Universal Robots PolyScope program: a_full_bow.urp

Program a_full_bow (installation=string_planes directory=/programs createdIn=5.17.3 lastSavedIn=5.17.3 robotSerialNumber=20245501435)
Calibrated DH parameters: a=[0.000154, -0.137004, -0.385524, -0.00002, 0.000092, 0]; d=[0.162441, 211.794786, -230.585024, 18.923638, 0.099786, 0.09951]; alpha=[1.569493, -0.001902, 0.003874, 1.570111, -1.570167, 0]; deltaTheta=[0, -1.242934, 1.056292, 0.186646, 0.000002, 0.000001]
InitVariablesNode
Robot Program (runOnlyOnce=false)
  bow_dir := False
  note_dur := 3
  Timer (action=Start) variable(name=timer_1)
  If bow_dir
    MoveL speed 250 mm/s, acceleration 1200 mm/s^2 (useActiveTCP=true) feature=Base
      Waypoint Waypoint_2: TCP in base x=374.969 y=359.127 z=303.035 mm, rx=1.6275 ry=2.3373 rz=-1.1146 rad; joints [-156.117, -66.368, 101.552, -88.734, -114.429, -168.118] deg; TCP offset x=28.21 y=-96.107 z=-99.69 mm, rx=0 ry=0 rz=0 rad
        Until EXPRESSION (allowActions=false) ExpressionBranch=timer_1≟note_dur
  Else 
    MoveL speed 250 mm/s, acceleration 1200 mm/s^2 (useActiveTCP=true) feature=Base
      Waypoint Waypoint_1: TCP in base x=277.237 y=734.032 z=156.892 mm, rx=1.7389 ry=2.3104 rz=-1.1078 rad; joints [-126.647, -28.123, 54.729, -74.616, -91.964, -141.812] deg; TCP offset x=28.21 y=-96.107 z=-99.69 mm, rx=0 ry=0 rz=0 rad
        Until EXPRESSION (allowActions=false) ExpressionBranch=timer_1≟note_dur
  SuppressedNode
    MoveL speed 250 mm/s, acceleration 1200 mm/s^2 (useActiveTCP=true) feature=Base
      Waypoint Waypoint_1: TCP in base x=277.237 y=734.032 z=156.892 mm, rx=1.7389 ry=2.3104 rz=-1.1078 rad; joints [-126.647, -28.123, 54.729, -74.616, -91.964, -141.812] deg
      Waypoint Waypoint_3: motionParameters(blendRadius=0.05); TCP in base x=335.809 y=527.638 z=230.762 mm, rx=1.7389 ry=2.3104 rz=-1.1078 rad; joints [-141.244, -51.172, 87.867, -86.053, -101.589, -152.842] deg; TCP offset x=28.21 y=-96.107 z=-99.69 mm, rx=0 ry=0 rz=0 rad
      Waypoint Waypoint_2: TCP in base x=393.128 y=325.659 z=303.053 mm, rx=1.7389 ry=2.3104 rz=-1.1078 rad; joints [-160.523, -67.347, 103.242, -90.17, -113.569, -168.748] deg
  Timer (action=Stop) variable=timer_1
  Timer (action=Reset) variable=timer_1
